// TIA Portal V16 export
// export: Created 2024-05-10T06:46:42.9789844Z, ExportSetting WithDefaults, DisplayName Totally Integrated Automation Portal, DisplayVersion V16, DisplayName TIA Portal Version Control Interface, DisplayVersion V16, DisplayName TIA Portal Openness, DisplayVersion V16, DisplayName STEP 7 Professional, DisplayVersion V16, DisplayName STEP 7 Safety, DisplayVersion V16, DisplayName WinCC Professional, DisplayVersion V16
FUNCTION_BLOCK "F110_Inv"   // FB110, LAD
{ S7_Optimized_Access := 'TRUE' }
VERSION : 0.1
// 变频器FB
// stored: AutoNumber false, IsIECCheckEnabled false, IsRetainMemResEnabled false, MemoryReserve 100, SetENOAutomatically false, UDAEnableTagReadback false
   VAR_INPUT
      I_AutoAdv : Bool;   // 自动正转指令
      I_AutoRet : Bool;   // 自动反转指令
      I_ManAdv : Bool;   // 手动正转指令
      I_ManRet : Bool;   // 手动反转指令
      I_AdvCond : Bool;   // 正转动作条件
      I_RetCond : Bool;   // 反转动作条件
      I_AdvLS : Bool;   // 正转到位
      I_RetLS : Bool;   // 反转到位
      I_AdLowP : Bool;   // 正转减速位置
      I_ReLowP : Bool;   // 反转减速位置
      I_InvNorm : Bool;   // 变频器正常
      I_InvCut : Bool;   // 变频器切断
      IW_ChkTim : Time;   // 动作确认时间
      I_FoBrRel : Bool;   // 刹车强制解除
      I_Rest : Bool;   // 异常复位
      I_ManMode : Bool;   // 手动模式
   END_VAR
   VAR_OUTPUT
      Q_AdvEnd : Bool;   // 正转到位
      Q_RetEnd : Bool;   // 反转到位
      O_AdvRot : Bool;   // 正转
      O_RetRot : Bool;   // 反转
      O_HiSpeed : Bool;   // 高速
      O_LoSpeed { ExternalVisible := 'False'} : Bool;   // 低速
      O_InvRes : Bool;   // INV.复位输出
      O_InvStop : Bool;   // INV.输出正常
      O_BrRel : Bool;   // 制动器解除输出
      O_LS_Flt : Bool;   // LS异常
      O_ActFlt : Bool;   // 动作异常
      O_InvFlt : Bool;   // 变频器异常
   END_VAR
   VAR
      MT_ActF : IEC_TIMER;   // 动作异常
   END_VAR
   VAR_TEMP
      M_MoveOK : Bool;   // 动作可
      M_AdvM : Bool;   // 正转操作
      M_RetM : Bool;   // 反转操作
      M_AdvComm : Bool;   // 正转指示
      M_RetComm : Bool;   // 反转指示
      M_TimOf : Bool;   // 动作无效确认
   END_VAR
   VAR_TEMP   // added for the SCL form of the ladder/FBD networks
      _w1 : Bool;
   END_VAR
BEGIN

REGION Network 1: 动作无效确认
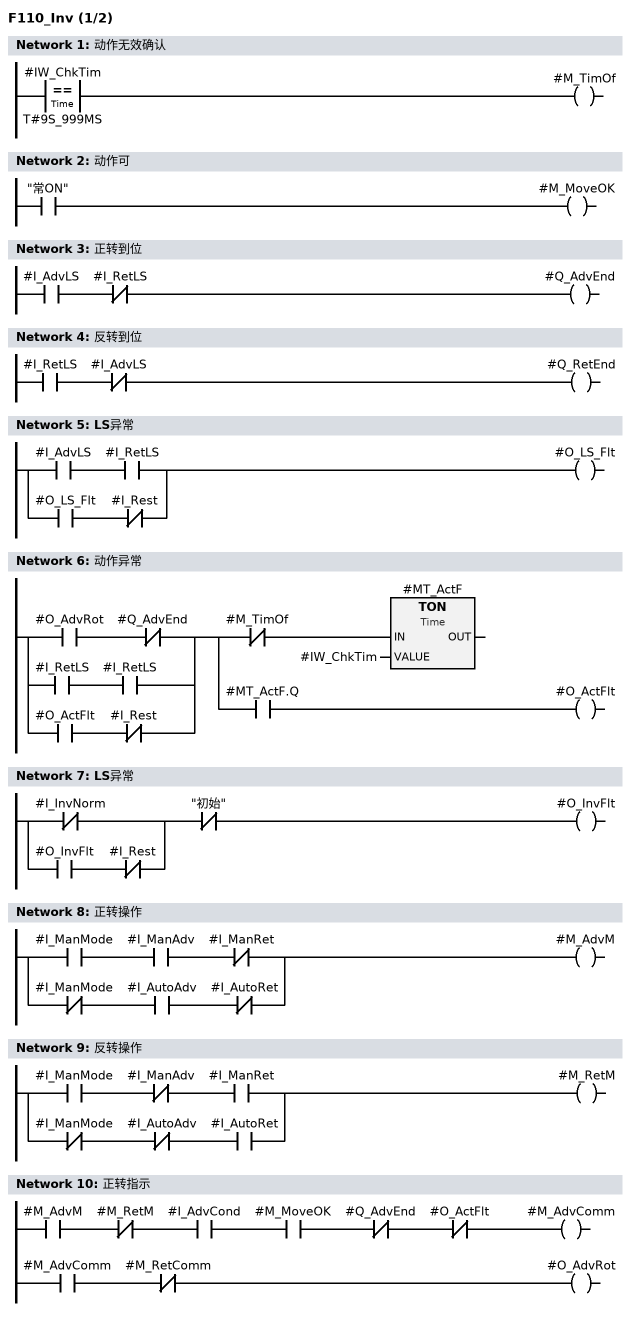
   RUNG wire#powerrail
      { S7_Templates := "SrcType := Time" } EQ_Contact(in1 := #IW_ChkTim, in2 := T#9S_999MS)
      Coil( #M_TimOf )
   END_RUNG
   // the same network as SCL:
   #M_TimOf := #IW_ChkTim = T#9S_999MS;
END_REGION

REGION Network 2: 动作可
   RUNG wire#powerrail
      Contact( "常ON" )
      Coil( #M_MoveOK )
   END_RUNG
   // the same network as SCL:
   #M_MoveOK := "常ON";
END_REGION

REGION Network 3: 正转到位
   RUNG wire#powerrail
      Contact( #I_AdvLS )
      I_Contact( #I_RetLS )
      Coil( #Q_AdvEnd )
   END_RUNG
   // the same network as SCL:
   #Q_AdvEnd := #I_AdvLS AND NOT #I_RetLS;
END_REGION

REGION Network 4: 反转到位
   RUNG wire#powerrail
      Contact( #I_RetLS )
      I_Contact( #I_AdvLS )
      Coil( #Q_RetEnd )
   END_RUNG
   // the same network as SCL:
   #Q_RetEnd := #I_RetLS AND NOT #I_AdvLS;
END_REGION

REGION Network 5: LS异常
   RUNG wire#powerrail
      Contact( #I_AdvLS )
      Contact( #I_RetLS )
      wire#w1
      Coil( #O_LS_Flt )
   END_RUNG
   RUNG wire#powerrail
      Contact( #O_LS_Flt )
      I_Contact( #I_Rest )
   END_RUNG wire#w1
   // the same network as SCL:
   #O_LS_Flt := (#I_AdvLS AND #I_RetLS) OR (#O_LS_Flt AND NOT #I_Rest);
END_REGION

REGION Network 6: 动作异常
   #_w1 := (#O_AdvRot AND NOT #Q_AdvEnd) OR (#I_RetLS AND #I_RetLS) OR (#O_ActFlt AND NOT #I_Rest);
   #MT_ActF.TON(IN := #_w1 AND NOT #M_TimOf, PT := #IW_ChkTim);   // TON coil
   #O_ActFlt := #_w1 AND #MT_ActF.Q;
END_REGION

REGION Network 7: LS异常
   RUNG wire#powerrail
      I_Contact( #I_InvNorm )
      wire#w1
      I_Contact( "初始" )
      Coil( #O_InvFlt )
   END_RUNG
   RUNG wire#powerrail
      Contact( #O_InvFlt )
      I_Contact( #I_Rest )
   END_RUNG wire#w1
   // the same network as SCL:
   #O_InvFlt := (NOT #I_InvNorm OR (#O_InvFlt AND NOT #I_Rest)) AND NOT "初始";
END_REGION

REGION Network 8: 正转操作
   RUNG wire#powerrail
      Contact( #I_ManMode )
      Contact( #I_ManAdv )
      I_Contact( #I_ManRet )
      wire#w1
      Coil( #M_AdvM )
   END_RUNG
   RUNG wire#powerrail
      I_Contact( #I_ManMode )
      Contact( #I_AutoAdv )
      I_Contact( #I_AutoRet )
   END_RUNG wire#w1
   // the same network as SCL:
   #M_AdvM := (#I_ManMode AND #I_ManAdv AND NOT #I_ManRet) OR (NOT #I_ManMode AND #I_AutoAdv AND NOT #I_AutoRet);
END_REGION

REGION Network 9: 反转操作
   RUNG wire#powerrail
      Contact( #I_ManMode )
      I_Contact( #I_ManAdv )
      Contact( #I_ManRet )
      wire#w1
      Coil( #M_RetM )
   END_RUNG
   RUNG wire#powerrail
      I_Contact( #I_ManMode )
      I_Contact( #I_AutoAdv )
      Contact( #I_AutoRet )
   END_RUNG wire#w1
   // the same network as SCL:
   #M_RetM := (#I_ManMode AND NOT #I_ManAdv AND #I_ManRet) OR (NOT #I_ManMode AND NOT #I_AutoAdv AND #I_AutoRet);
END_REGION

REGION Network 10: 正转指示
   RUNG wire#powerrail
      Contact( #M_AdvM )
      I_Contact( #M_RetM )
      Contact( #I_AdvCond )
      Contact( #M_MoveOK )
      I_Contact( #Q_AdvEnd )
      I_Contact( #O_ActFlt )
      Coil( #M_AdvComm )
   END_RUNG
   RUNG wire#powerrail
      Contact( #M_AdvComm )
      I_Contact( #M_RetComm )
      Coil( #O_AdvRot )
   END_RUNG
   // the same network as SCL:
   #M_AdvComm := #M_AdvM AND NOT #M_RetM AND #I_AdvCond AND #M_MoveOK AND NOT #Q_AdvEnd AND NOT #O_ActFlt;
   #O_AdvRot := #M_AdvComm AND NOT #M_RetComm;
END_REGION

REGION Network 11: 反转指示
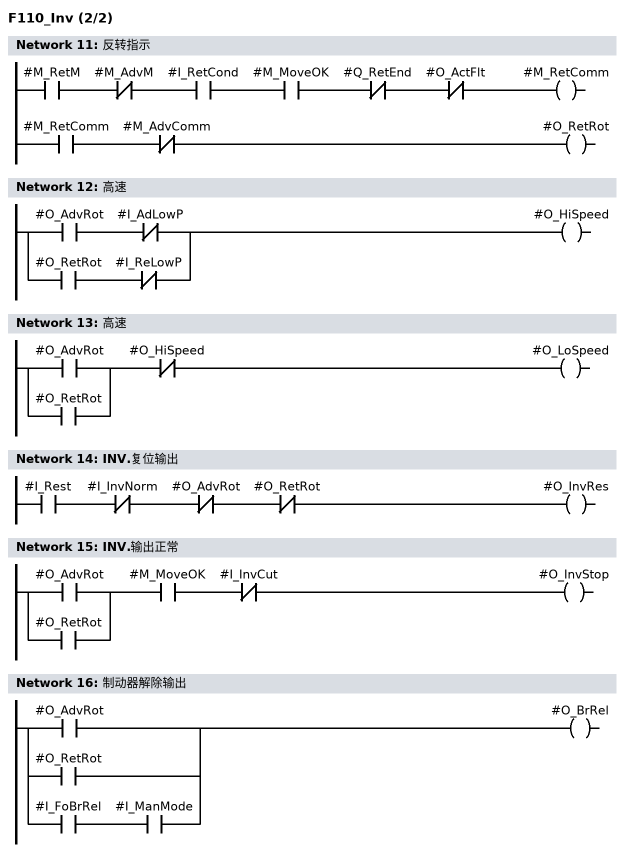
   RUNG wire#powerrail
      Contact( #M_RetM )
      I_Contact( #M_AdvM )
      Contact( #I_RetCond )
      Contact( #M_MoveOK )
      I_Contact( #Q_RetEnd )
      I_Contact( #O_ActFlt )
      Coil( #M_RetComm )
   END_RUNG
   RUNG wire#powerrail
      Contact( #M_RetComm )
      I_Contact( #M_AdvComm )
      Coil( #O_RetRot )
   END_RUNG
   // the same network as SCL:
   #M_RetComm := #M_RetM AND NOT #M_AdvM AND #I_RetCond AND #M_MoveOK AND NOT #Q_RetEnd AND NOT #O_ActFlt;
   #O_RetRot := #M_RetComm AND NOT #M_AdvComm;
END_REGION

REGION Network 12: 高速
   RUNG wire#powerrail
      Contact( #O_AdvRot )
      I_Contact( #I_AdLowP )
      wire#w1
      Coil( #O_HiSpeed )
   END_RUNG
   RUNG wire#powerrail
      Contact( #O_RetRot )
      I_Contact( #I_ReLowP )
   END_RUNG wire#w1
   // the same network as SCL:
   #O_HiSpeed := (#O_AdvRot AND NOT #I_AdLowP) OR (#O_RetRot AND NOT #I_ReLowP);
END_REGION

REGION Network 13: 高速
   RUNG wire#powerrail
      Contact( #O_AdvRot )
      wire#w1
      I_Contact( #O_HiSpeed )
      Coil( #O_LoSpeed )
   END_RUNG
   RUNG wire#powerrail
      Contact( #O_RetRot )
   END_RUNG wire#w1
   // the same network as SCL:
   #O_LoSpeed := (#O_AdvRot OR #O_RetRot) AND NOT #O_HiSpeed;
END_REGION

REGION Network 14: INV.复位输出
   RUNG wire#powerrail
      Contact( #I_Rest )
      I_Contact( #I_InvNorm )
      I_Contact( #O_AdvRot )
      I_Contact( #O_RetRot )
      Coil( #O_InvRes )
   END_RUNG
   // the same network as SCL:
   #O_InvRes := #I_Rest AND NOT #I_InvNorm AND NOT #O_AdvRot AND NOT #O_RetRot;
END_REGION

REGION Network 15: INV.输出正常
   RUNG wire#powerrail
      Contact( #O_AdvRot )
      wire#w1
      Contact( #M_MoveOK )
      I_Contact( #I_InvCut )
      Coil( #O_InvStop )
   END_RUNG
   RUNG wire#powerrail
      Contact( #O_RetRot )
   END_RUNG wire#w1
   // the same network as SCL:
   #O_InvStop := (#O_AdvRot OR #O_RetRot) AND #M_MoveOK AND NOT #I_InvCut;
END_REGION

REGION Network 16: 制动器解除输出
   RUNG wire#powerrail
      Contact( #O_AdvRot )
      wire#w1
      Coil( #O_BrRel )
   END_RUNG
   RUNG wire#powerrail
      Contact( #O_RetRot )
   END_RUNG wire#w1
   RUNG wire#powerrail
      Contact( #I_FoBrRel )
      Contact( #I_ManMode )
   END_RUNG wire#w1
   // the same network as SCL:
   #O_BrRel := #O_AdvRot OR #O_RetRot OR (#I_FoBrRel AND #I_ManMode);
END_REGION
END_FUNCTION_BLOCK
